{region '#Template'}
	{attribute 'Version' := '5.0.1.0'}
	{attribute 'Tags' := '"LCID": "1031", "Text": "Universal, Control, PID, Loop"'}
	{attribute 'Tags' := '"LCID": "1033", "Text": "Universal, Control, PID, Loop"'}
	{attribute 'Using' := '"Type": "Template", "URI": "BA2_Param"'}
	{attribute 'Description' := '"LCID": "1031", "Text": "Regler mit Sollwert Object"'}
	{attribute 'Description' := '"LCID": "1033", "Text": "Controller with setpoint object"'}
{endregion}
FUNCTION_BLOCK FB_BA_PID_Sp EXTENDS FB_BA_View
VAR_INPUT
	bEn						: BOOL;
	fX						: REAL;
	bSync					: BOOL;
	fSync					: REAL;
END_VAR
VAR_OUTPUT
	fY						: REAL;
	fMax					: REAL;
	fMin					: REAL;	
END_VAR
VAR_INPUT CONSTANT
	Sp						: FB_BA_AV_Op;		 
	Ctrl					: FB_BA_Loop;	
END_VAR

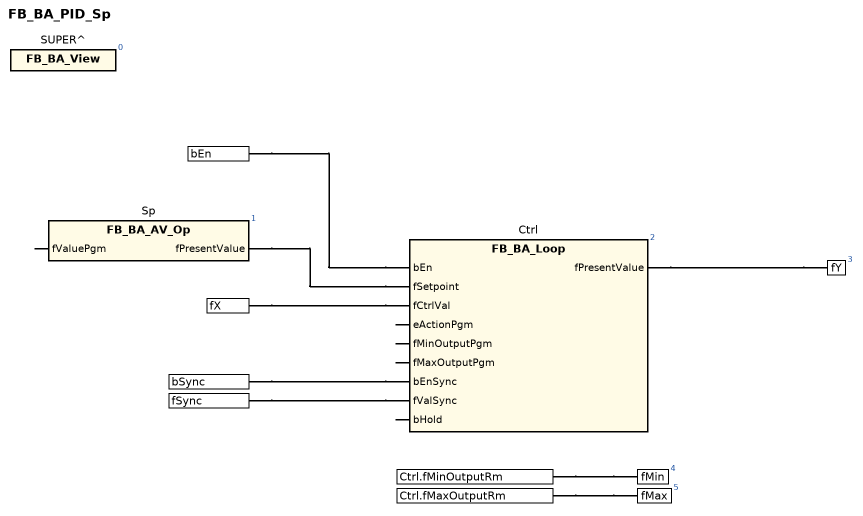
SUPER^(); // FB_BA_View
Sp(); // FB_BA_AV_Op
Ctrl(bEn := bEn, fSetpoint := Sp.fPresentValue, fCtrlVal := fX, bEnSync := bSync, fValSync := fSync); // FB_BA_Loop
fY := Ctrl.fPresentValue;
fMin := Ctrl.fMinOutputRm;
fMax := Ctrl.fMaxOutputRm;

METHOD FB_init : BOOL
VAR_INPUT
	bInitRetains : BOOL; // if TRUE, the retain variables are initialized (warm start / cold start)
	bInCopyCode : BOOL;  // if TRUE, the instance afterwards gets moved into the copy code (online change)
END_VAR
Sp.iParent					:= THIS^;
Sp.iLabel					:= LblFun_Setpoint;   					 	 
Sp.eUnit 					:= E_BA_Unit.eTemperature_DegreesCelsius;								 
Sp.fValueRm					:= 21.0;															 
Sp.fCOVIncrement			:= BA2_Param.fDefCOVIncrement;

Ctrl.iParent				:= THIS^;
Ctrl.iLabel					:= LblFun_LoopObject;  
Ctrl.eOpMode				:= E_BA_PIDMode.ePID;								 	 										 
Ctrl.eOutputUnit			:= E_BA_Unit.eOther_Percent;
Ctrl.eActionRm				:= E_BA_Action.eReverse;
Ctrl.fProportionalConstant	:= 3;
Ctrl.fIntegralConstant		:= 180;
Ctrl.fDerivativeConstant	:= 0;
Ctrl.fMaxOutputRm 			:= 100;
Ctrl.fMinOutputRm			:= 0;
Ctrl.fCOVIncrement			:= 0;
Ctrl.nDampConstant			:= 0;
Ctrl.fNeutralZone			:= 0;
END_METHOD

END_FUNCTION_BLOCK

(* stored: Version 1.1.0.1, ProductVersion 3.1.4024.15
   POU FB_BA_PID_Sp: Id {79266ebd-dce2-4431-a546-e1ebc7ff4dd5}, SpecialFunc None
   Method FB_init: Id {3386f0f2-178d-4227-a45d-7737d5736a7c} *)
